INTERFACE I_Queue EXTENDS I_Collection

METHOD PUBLIC Enqueue
VAR_INPUT
	Item : ANY;
END_VAR
END_METHOD

METHOD PUBLIC TryDequeue : BOOL;
VAR_INPUT
	Destination : ANY;
END_VAR
END_METHOD

METHOD PUBLIC TryPeek : BOOL;
VAR_INPUT
	Destination : ANY;
END_VAR
END_METHOD

END_INTERFACE

(* stored: Version 1.1.0.1, ProductVersion 3.1.4024.12
   Itf I_Queue: Id {09b3322b-c832-090a-1623-e3f7735cbe68}
   Method Enqueue: Id {3fa5d10e-cd5f-0481-38a0-020258383a83}
   Method TryDequeue: Id {a35d87d9-3b0a-095e-1451-845334d474da}
   Method TryPeek: Id {f7be56f0-d686-0ac6-2fc3-a0a70ee864a4} *)
